PROGRAM MAIN
VAR
	IPAdress		: STRING 	:= '10.0.120.102';
	Port			: UINT		:= 8080;
	UpdatePeriod	: TIME		:= T#60s;
	fbHttpProcess	: FB_IotHttpClient :=(	sHostName			:= IPAdress,
								  			bKeepAlive			:= TRUE, 
											tConnectionTimeout	:= T#10S);
	fbProcessPost	: FB_EventHTTP_Post;
	
	HttpSend		: BOOL := FALSE;
	
	API_Msg			: STRING[255] := '';
	bSuccess		: BOOL;
	bError			: BOOL;
	
END_VAR


IF NOT fbHttpProcess.bConfigured THEN 
	fbHttpProcess.nHostPort 				:= Port;
	fbHttpProcess.stTLS.bNoServerCertCheck 	:= TRUE;
END_IF

IF fbHttpProcess.bConfigured THEN 
	fbProcessPost( 	bSend		:= HttpSend, 
				 	fbClient	:= fbHttpProcess, 
					API_URI		:= '/hello?data=123',
				 	API_Msg 	:= API_Msg,
					bSuccess 	=> bSuccess,
					bError		=> bError );
END_IF 

fbHttpProcess.Execute();

END_PROGRAM

(* stored: Version 1.1.0.1, ProductVersion 3.1.4024.12
   POU MAIN: Id {41d800dd-6c26-40c4-8b1f-d3de318c5d3b}, SpecialFunc None *)
